// TwinCAT 3 PLC project Oefening3
// ProgramVersion: 3.1.4023.0
// libraries:
//   Tc2_BABasic, * (Beckhoff Automation GmbH)
//   Tc2_Standard, * (Beckhoff Automation GmbH)
//   Tc2_System, * (Beckhoff Automation GmbH)
//   Tc2_Utilities, * (Beckhoff Automation GmbH)
//   Tc3_Module, * (Beckhoff Automation GmbH)
// project tree:
//   / GlobalTextList.TcGTLO, PlcTask.TcTTO, Visualization Manager.TcVMO (not stored)
//   POUs/ FB_Knipperlicht.TcPOU, MAIN.TcPOU
//   VISUs/ Oefening3_VISU.TcVIS
// (motion and I/O tree: see PLC project oefening1)
// real-time tasks:
//   TASK PlcTask: cycle T#10ms, priority 20, ADS port 350
//   TASK PlcTask1: cycle T#10ms, priority 21, ADS port 351
//   TASK PlcTask2: cycle T#10ms, priority 22, ADS port 352
//   TASK PlcTask3: cycle T#10ms, priority 23, ADS port 353
//   TASK PlcTask4: cycle T#10ms, priority 24, ADS port 354
//   TASK PlcTask5: cycle T#10ms, priority 25, ADS port 355

CONFIGURATION Oefening3
    RESOURCE PLC ON TwinCAT3
        TASK PlcTask(INTERVAL := T#10ms, PRIORITY := 23);
        PROGRAM MAIN WITH PlcTask : MAIN;
    END_RESOURCE
END_CONFIGURATION

// ---- POUs/MAIN.TcPOU
PROGRAM MAIN

VAR_INPUT
	requestedTemp : INT;
	actualTemp : INT;
END_VAR

VAR_OUTPUT
END_VAR

VAR
	verwarming : BOOL;
	
	Knipperlicht : FB_Knipperlicht;
	i: INT;
	
	FB_LocalSystemTime : FB_LocalSystemTime;
	FB_WeeklyTimeSwitch : FB_WeeklyTimeSwitch;
	
	OneSecondCount : BOOL;
	tempUpdate : ARRAY [1..20] OF INT;
	F_TRIG : F_TRIG;
	//YEAR: STRING;
	//MONTH: STRING;
	//DAY: STRING;
	//HOUR: STRING;
	//MINUTE: STRING;
	//SECOND: STRING;
	TIMESTAMP: DATE_AND_TIME;
END_VAR

FB_LocalSystemTime(bEnable:= TRUE);


//YEAR := WORD_TO_STRING(FB_LocalSystemTime.systemTime.wYear);
//MONTH := WORD_TO_STRING(FB_LocalSystemTime.systemTime.wMonth);
//DAY := WORD_TO_STRING(FB_LocalSystemTime.systemTime.wDay);
//HOUR := WORD_TO_STRING(FB_LocalSystemTime.systemTime.wHour);
//MINUTE := WORD_TO_STRING(FB_LocalSystemTime.systemTime.wMinute);
//SECOND := WORD_TO_STRING(FB_LocalSystemTime.systemTime.wSecond);	
//TIMESTAMP := CONCAT('DT#', YEAR);
//TIMESTAMP := CONCAT(TIMESTAMP , '-');
//TIMESTAMP := CONCAT(TIMESTAMP , MONTH);
//TIMESTAMP := CONCAT(TIMESTAMP , '-');
//TIMESTAMP := CONCAT(TIMESTAMP , DAY);
//TIMESTAMP := CONCAT(TIMESTAMP , '-');
//TIMESTAMP := CONCAT(TIMESTAMP , HOUR);
//TIMESTAMP := CONCAT(TIMESTAMP , ':');
//TIMESTAMP := CONCAT(TIMESTAMP , MINUTE);
//TIMESTAMP := CONCAT(TIMESTAMP , ':');
//TIMESTAMP := CONCAT(TIMESTAMP , SECOND);

TIMESTAMP := SYSTEMTIME_TO_DT(TIMESTR:= FB_LocalSystemTime.systemTime);

FB_WeeklyTimeSwitch(
	bEnable:= TRUE, 
	tCurrentDateTime:= TIMESTAMP,//FB_LocalSystemTime.systemTime, 
	tSwitchOnTime:= TOD#08:00, 
	tSwitchOffTime:= TOD#20:00, 
	bSunday:= TRUE, 
	bMonday:= TRUE, 
	bTuesday:= TRUE, 
	bWednesday:= TRUE, 
	bThursday:= TRUE, 
	bFriday:= TRUE, 
	bSaturday:= TRUE);	
	
IF FB_WeeklyTimeSwitch.bOutput THEN
	IF (actualTemp < requestedTemp) THEN
		verwarming := TRUE;
	ELSE
		verwarming := FALSE;
	END_IF
ELSE
	verwarming := FALSE;
END_IF

Knipperlicht(Enable:= TRUE, OnTime:= T#1S, OfTime:= T#0S, Q=> OneSecondCount);
F_TRIG(CLK:= Knipperlicht.Q);

IF F_TRIG.Q THEN
	IF i <= 20 THEN;
		tempUpdate[i+1] := actualTemp;
		i := i + 1;
	ELSE
		i := 0;
	END_IF
END_IF

END_PROGRAM

// ---- POUs/FB_Knipperlicht.TcPOU
FUNCTION_BLOCK FB_Knipperlicht
VAR_INPUT
	Enable : BOOL;	(* activatie knipperlicht*)
	OnTime : TIME;  (* tijd dat de lamp aan is *)
	OfTime : TIME;  (* tijd dat de lamp uit is *)
	CyclesReset : BOOL;
END_VAR

VAR_OUTPUT
	Q: BOOL;		(* het knipperlicht *)
	Freq: REAL;		(* de knipperfrequentie *)
	Duty: REAL;     (* de verhouding aan/totale-tijd *)
	Cycles: INT;	(* Hoeveelheid cycles voltooid *)
END_VAR

VAR
	Counter : BOOL;
	R_TRIG : R_TRIG;
	tOnTime: TOF;
	tOfTime: TON;
	tTotalTime: TIME; 
END_VAR

IF Enable THEN
	IF CyclesReset THEN
		Cycles := 0;
	ELSE
	tTotalTime := OnTime + OfTime;
	Duty := (TIME_TO_REAL(OnTime)/(TIME_TO_REAL(OnTime)+TIME_TO_REAL(OfTime))*100);
	Freq := 1000 / (TIME_TO_REAL(OnTime)+TIME_TO_REAL(OfTime));
	
	tOnTime(IN:= NOT tOfTime.Q  , PT:= OnTime, Q=>Q);
	tOfTime(IN:= tOntime.Q 	    , PT:= OfTime, Q=>Q);
	
	R_TRIG(CLK:= Q, Q=> Counter);
	Cycles := Cycles + BOOL_TO_INT(Counter);
	END_IF
ELSE
	Q := FALSE;
END_IF

END_FUNCTION_BLOCK

// ---- VISUs/Oefening3_VISU.TcVIS
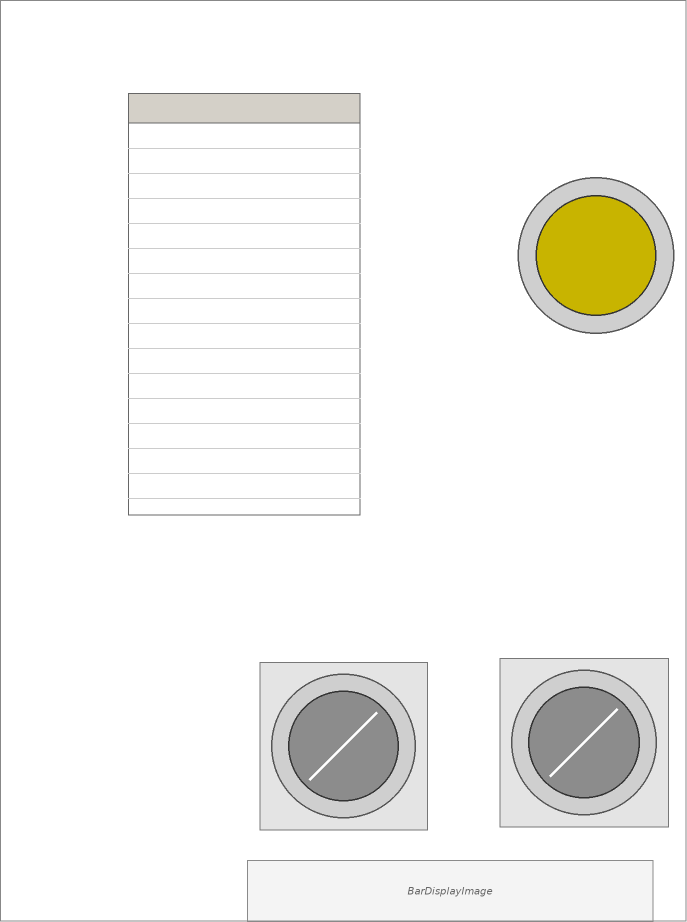
VISUALIZATION Oefening3_VISU  // 687x922
    Potentiometer360 (230,662 227x168), variable: MAIN.requestedTemp, style: Potentiometer-Potentiometer360-Gray, scale format: %.1f, scale 10..30
        p2431819421: Outside
    Potentiometer360 (497,658 174x169), variable: MAIN.actualTemp, style: Potentiometer-Potentiometer360-Gray, scale format: %.1f, scale -30..40
        p2431819421: Outside
    BarDisplayImage (247,860 406x62), value: MAIN.actualTemp, style: BarDisplayImage-Gray, scale format: %.1f, scale 0..100
    Lamp1 (505,135 182x241), variable: MAIN.verwarming, style: Lamp-Lamp1-Yellow
    Table (128,93 232x422), data array: MAIN.tempUpdate
        p3854506369: MAIN.tempUpdate[INDEX]
END_VISUALIZATION
